ADAPTER PLCnextBusAdapter
  (* Standard: 61499-2; Description: Copyright (c) 2022 Peirlberger Juergen This program and the accompanying materials are made available under the terms of the Eclipse Public License 2.0 which is available at https://www.eclipse.org/legal/epl-2.0/ SPDX-License-Identifier: EPL-2.0 Copyright (c) 2022 Peirlberger Juergen. This program and the accompanying materials are made available under the terms of the Eclipse Public License 2.0 which is available at http://www.eclipse.org/legal/epl-2.0. SPDX-License-Identifier: EPL-2.0 *)
  (* Version 1.0, 2022-04-07, Peirlberger Juergen *)
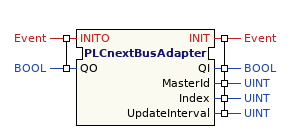
  EVENT_INPUT
    INITO WITH QO; (* Initialization Confirm *)
  END_EVENT
  EVENT_OUTPUT
    INIT WITH Index, UpdateInterval, MasterId, QI; (* Service Initialization *)
  END_EVENT
  VAR_INPUT
    QO : BOOL;
  END_VAR
  VAR_OUTPUT
    QI : BOOL;
    MasterId : UINT;
    Index : UINT;
    UpdateInterval : UINT; (* Global update interval of slave modules in Hz *)
  END_VAR
  SERVICE SOCKET/PLUG
    SEQUENCE request_confirm
      SOCKET.REQ(REQD) -> PLUG.REQ(REQD);
      PLUG.CNF(CNFD) -> SOCKET.CNF(CNFD);
    END_SEQUENCE
    SEQUENCE indication_response
      PLUG.IND(INDD) -> SOCKET.IND(INDD);
      SOCKET.RSP(RSPD) -> PLUG.RSP(RSPD);
    END_SEQUENCE
  END_SERVICE
END_ADAPTER
